// Mitsubishi GX Works2 project: 6.14 finsh   PLC: FX3G

// global labels: Global1
VAR_GLOBAL
  sw7_startday AT X007 : BOOL;
  output7_light AT Y007 : BOOL;
  sw5_emrgency AT X005 : BOOL;
  raw_matirial_end AT M1 : BOOL;
  matirial_end AT M1 : BOOL;
  output5_light AT M7 : BOOL;
  work_day_m5 AT M5 : BOOL;
  lamf_work_day AT Y007 : BOOL;
  Petel_input_amount AT D1148 : REAL;
  Petel_cornt_amount AT D1250 : REAL;
  Limonl_input_amount AT D1195 : REAL;
  Gomi_input_amount AT D1245 : REAL;
  Gomi_cornt_amount AT D1270 : REAL;
  Meatzv_input_amount AT D1295 : REAL;
  Meyatzev_input_amount AT D1295 : REAL;
  Meyatzev_cornt_amount AT D1300 : REAL;
  output AT D8282 : INT;
  start_ice_crem AT X001 : BOOL;
  timer_icecream5 AT TC1 : BOOL;
END_VAR
VAR_GLOBAL CONSTANT
  Sec_icecream : INT := K50;
END_VAR
VAR_GLOBAL
  start_icecream AT X001 : BOOL;
  Petel_ragil_help AT M52 : BOOL;
  Petel_pinoc_help AT M53 : BOOL;
  Limon_ragil_help AT M54 : BOOL;
  Limon_input_amount AT D1195 : REAL;
  Limon_cornt_amount AT D1200 : REAL;
  Limon_pinoc_help AT M55 : BOOL;
  Petel_ragil AT M22 : BOOL;
  Petel_pinoc AT M23 : BOOL;
  Limon_ragil AT M24 : BOOL;
  Limon_pinoc AT M25 : BOOL;
  lamp_y2 AT Y002 : BOOL;
END_VAR
VAR_GLOBAL CONSTANT
  division_constant : REAL := 400;
END_VAR
VAR_GLOBAL
  analog_input_1 AT D8280 : INT;
  goomigum_type AT D1502 : REAL;
  Min_regular AT E0.0 : REAL;
  Max_regular AT E5.0 : REAL;
  Min_pinuk AT E6.0 : REAL;
  check_inventory AT M20 : BOOL;
  choose_regular AT M300 : BOOL;
  choose_pinuk AT M400 : BOOL;
END_VAR
VAR_GLOBAL CONSTANT
  const280 : REAL := 280;
  const_280 : REAL := 280;
  conat_35 : REAL := 280;
  const_35 : REAL := 35;
END_VAR
VAR_GLOBAL
  not_petel_ragil AT M61 : BOOL;
END_VAR
VAR_GLOBAL CONSTANT
  const_385 : REAL := 385;
  const_105 : REAL := 105;
  const_70 : REAL := 70;
  const_0 : REAL;
  const_420 : REAL := 420;
END_VAR
VAR_GLOBAL
  not_Petel_pinoc AT M62 : BOOL;
  not_Limon_ragil AT M63 : BOOL;
END_VAR
VAR_GLOBAL CONSTANT
  const_560 : REAL := 560;
END_VAR
VAR_GLOBAL
  not_Limon_pinoc AT M64 : BOOL;
END_VAR
VAR_GLOBAL CONSTANT
  const_140 : REAL := 140;
END_VAR
VAR_GLOBAL
  check_matirial AT M4 : BOOL;
  work : BOOL;
END_VAR
VAR_GLOBAL CONSTANT
  Five_Sec_icecream : INT := 50;
END_VAR
VAR_GLOBAL
  Time_icecream_finish AT TS1 : BOOL;
  is_making_icecream AT Y000 : BOOL;
  start_freeze AT X002 : BOOL;
END_VAR
VAR_GLOBAL CONSTANT
  const_700 : REAL := 700;
  const_490 : REAL := 490;
  const_350 : REAL := 350;
END_VAR
VAR_GLOBAL
  Premium_petel_icecream AT D1190 : REAL;
  Premium_lemonl_icecream AT D1210 : REAL;
  Regular_petel_icecream AT D1230 : REAL;
  Regular_lemonl_icecream AT D1240 : REAL;
END_VAR
VAR_GLOBAL CONSTANT
  const_8 : REAL := 8;
  const_10 : REAL;
END_VAR
VAR_GLOBAL
  sen_10 AT X003 : BOOL;
  lemf_y2 AT Y002 : BOOL;
  lamf_y2 AT Y002 : BOOL;
  Start_Packing AT X004 : BOOL;
  first_packing AT X000 : BOOL;
END_VAR
VAR_GLOBAL CONSTANT
  couter_seven_cones : INT := 7;
END_VAR
VAR_GLOBAL
  done_seven AT CC1 : BOOL;
  finish_seven AT CS1 : BOOL;
END_VAR
VAR_GLOBAL CONSTANT
  const_1 : INT := 1;
END_VAR
VAR_GLOBAL
  current_counter_cones AT CN1 : INT;
END_VAR
VAR_GLOBAL CONSTANT
  const_6_word : INT := 6;
END_VAR
VAR_GLOBAL
  lamp_y4 AT Y004 : BOOL;
  Amount_packages AT D1160 : REAL;
END_VAR
VAR_GLOBAL CONSTANT
  ADD_Package : REAL := 1;
END_VAR
VAR_GLOBAL
  end_day AT M10 : BOOL;
END_VAR
VAR_GLOBAL CONSTANT
  MUL40 : REAL := 40;
END_VAR
VAR_GLOBAL
  OutputMul AT D1170 : REAL;
  Frozen_premium_petel AT D3030 : REAL;
  Frozen_premium_lemon AT D3020 : REAL;
  Frozen_regular_petel AT D3040 : REAL;
  Frozen_regular_lemon AT D3060 : REAL;
  Stir_premium_petel AT D3080 : REAL;
  Stir_premium_lemon AT D4000 : REAL;
  Gummy_to_prod AT D5000 : REAL;
  Stir_regular_petel AT D4020 : REAL;
  Stir_regular_lemon AT D4040 : REAL;
END_VAR
VAR_GLOBAL CONSTANT
  const_28 : REAL := 28;
END_VAR
VAR_GLOBAL
  start_blink AT M60 : BOOL;
  timer_reset AT M0 : BOOL;
END_VAR
VAR_GLOBAL CONSTANT
  const_5 : INT := 50;
END_VAR
VAR_GLOBAL
  End_Timer1 AT TS1 : BOOL;
  Blink1 AT Y005 : BOOL;
  End_Timer2 AT TS2 : BOOL;
  Timer2 AT TC2 : BOOL;
  Blink2 AT Y006 : BOOL;
END_VAR
VAR_GLOBAL CONSTANT
  const_3 : INT := 30;
END_VAR
VAR_GLOBAL
  raw_materialsl_ferm AT D1165 : REAL;
  timer8 AT TC3 : BOOL;
  END_Timer3 AT TS3 : BOOL;
  ragil AT M30 : BOOL;
  ragi AT M22 : BOOL;
  pinoc AT M40 : BOOL;
  pinuk AT M40 : BOOL;
  regular AT M30 : BOOL;
  Ts5 AT Y005 : BOOL;
  ts6 AT Y006 : BOOL;
  ts7 AT Y007 : BOOL;
  ts4 AT Y004 : BOOL;
  lemon_icecream AT D1240 : REAL;
  petel_icecream AT D1230 : REAL;
  Frozen_petel AT D3030 : REAL;
  Frozen_lemon AT D3040 : REAL;
  lemonl_icecream AT D1210 : REAL;
END_VAR
VAR_GLOBAL CONSTANT
  const_2000 : REAL := 2000;
  const_80 : INT := 80;
END_VAR
VAR_GLOBAL
  Stir_petel AT D4030 : REAL;
  Stir_lemon AT D4040 : REAL;
  check666 AT X006 : BOOL;
  Timer4 AT TC4 : BOOL;
  End_Timer4 AT TS4 : BOOL;
  Timer800 AT TC10 : BOOL;
  End_Timer800 AT TS10 : BOOL;
  Timer5007 AT TC20 : BOOL;
  End_Timer5007 AT TS20 : BOOL;
  Timer5 AT TC30 : BOOL;
  Timer500 AT TC50 : BOOL;
  End_Timer500 AT TS50 : BOOL;
  End_Timer5 AT TS30 : BOOL;
  time_reset AT TC1 : BOOL;
END_VAR
VAR_GLOBAL CONSTANT
  stamtimer : INT := 10;
END_VAR
VAR_GLOBAL
  stammmm AT TC8 : BOOL;
  StAm AT TS8 : BOOL;
END_VAR
VAR_GLOBAL CONSTANT
  MUL400 : REAL := 400;
END_VAR
VAR_GLOBAL
  timer_pinuk AT TC55 : BOOL;
  timer_regular AT TC33 : BOOL;
  AD_matay1 AT TS33 : BOOL;
  AD_matay2 AT TS55 : BOOL;
END_VAR
VAR_GLOBAL CONSTANT
  const_imashelhazona : INT := 30;
END_VAR
VAR_GLOBAL
  regular_blink AT TS33 : BOOL;
  pinuk_blink AT TS55 : BOOL;
END_VAR
VAR_GLOBAL CONSTANT
  const_05 : INT := 5;
END_VAR
VAR_GLOBAL
  count_reset AT M20 : BOOL;
  count_reset11 AT TC8 : BOOL;
END_VAR
VAR_GLOBAL CONSTANT
  const_10a : INT := 10;
END_VAR
VAR_GLOBAL
  reset11a AT TS8 : BOOL;
  delete_frozen AT M39 : BOOL;
  Time_to_blink AT TC15 : BOOL;
END_VAR
VAR_GLOBAL CONSTANT
  const_6 : INT := 60;
END_VAR
VAR_GLOBAL
  Time_to_blink_f AT TS15 : BOOL;
  lamf_blink_help AT M70 : BOOL;
  fictive_1 AT TC11 : BOOL;
  fictive_2 AT TC12 : BOOL;
  fictive_1_help AT TS11 : BOOL;
  fictive_2_help AT TS12 : BOOL;
  Finish_blink AT M11 : BOOL;
END_VAR

// task Task_01 (event TRUE, interval 0, priority 31): POU_01

PROGRAM POU_01
(* structured ladder/FBD written out as ST: instructions are called as NAME(EN, inputs, outputs); _pN, _eN, _tN stand for wires *)
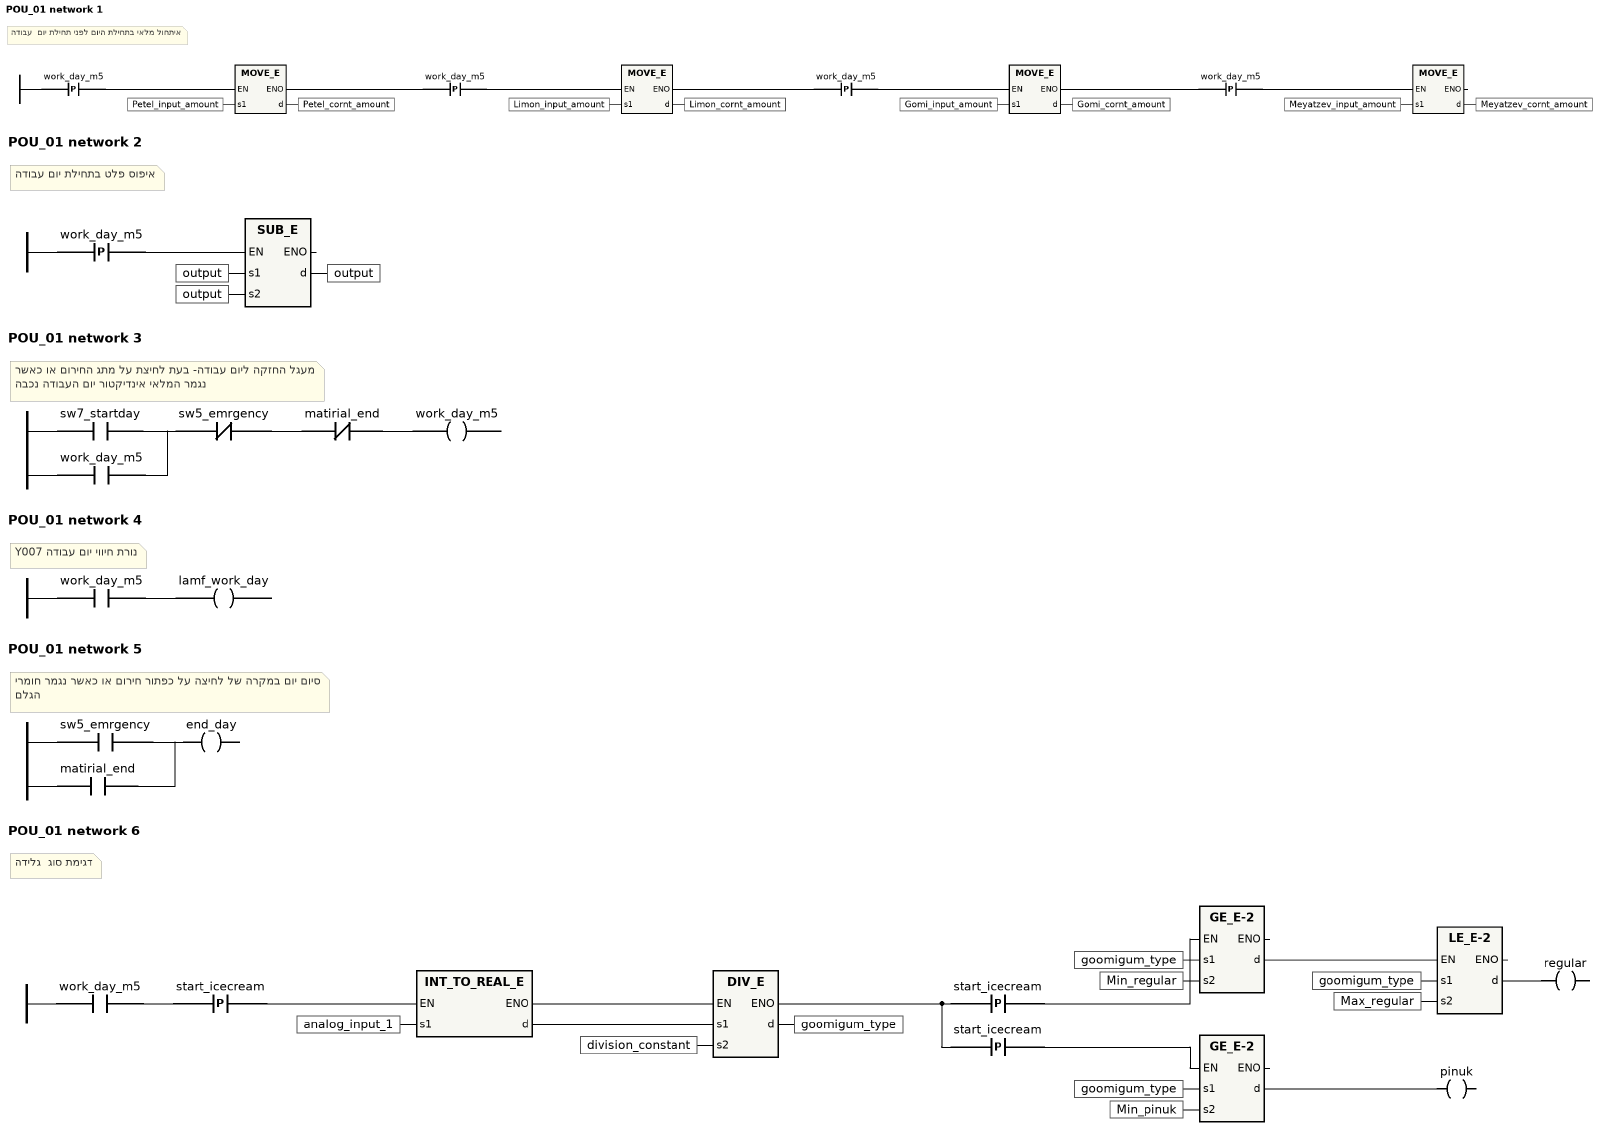
(* network 1 *)
(* איתחול מלאי בתחילת היום לפני תחילת יום  עבודה *)
_e1 := MOVE_E(LDP(TRUE, work_day_m5), Petel_input_amount, Petel_cornt_amount);
_e2 := MOVE_E(_e1 AND LDP(TRUE, work_day_m5), Limon_input_amount, Limon_cornt_amount);
_e3 := MOVE_E(_e2 AND LDP(TRUE, work_day_m5), Gomi_input_amount, Gomi_cornt_amount);
MOVE_E(_e3 AND LDP(TRUE, work_day_m5), Meyatzev_input_amount, Meyatzev_cornt_amount);
(* network 2 *)
(* איפוס פלט בתחילת יום עבודה *)
SUB_E(LDP(TRUE, work_day_m5), output, output, output);
(* network 3 *)
(* מעגל החזקה ליום עבודה- בעת לחיצת על מתג החירום או כאשר נגמר המלאי אינדיקטור יום העבודה נכבה *)
work_day_m5 := ((sw7_startday OR work_day_m5) AND NOT sw5_emrgency) AND NOT matirial_end;
(* network 4 *)
(* נורת חיווי יום עבודה Y007 *)
lamf_work_day := work_day_m5;
(* network 5 *)
(* סיום יום במקרה של לחיצה על כפתור חירום או כאשר נגמר חומרי הגלם *)
end_day := sw5_emrgency OR matirial_end;
(* network 6 *)
(* דגימת סוג  גלידה *)
_e2 := INT_TO_REAL_E(work_day_m5 AND LDP(TRUE, start_icecream), analog_input_1, _t1);
_e3 := DIV_E(_e2, _t1, division_constant, goomigum_type);
GE_E(_e3 AND LDP(TRUE, start_icecream), goomigum_type, Min_regular, _t4);
LE_E(_t4, goomigum_type, Max_regular, _t5);
regular := _t5;
GE_E(_e3 AND LDP(TRUE, start_icecream), goomigum_type, Min_pinuk, _t6);
pinuk := _t6;
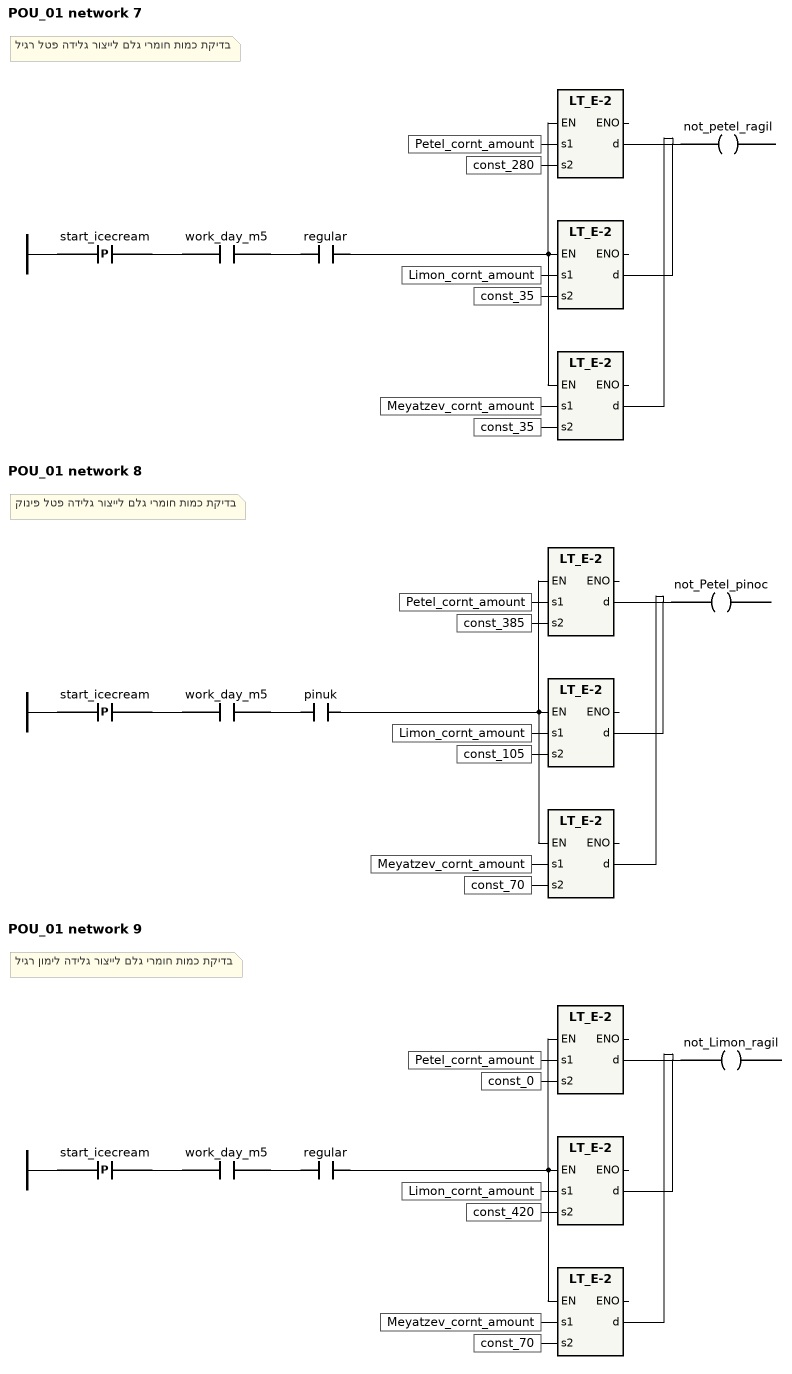
(* network 7 *)
(* בדיקת כמות חומרי גלם לייצור גלידה פטל רגיל *)
_p1 := LDP(TRUE, start_icecream) AND work_day_m5 AND regular;
LT_E(_p1, Petel_cornt_amount, const_280, _t2);
LT_E(_p1, Limon_cornt_amount, const_35, _t3);
LT_E(_p1, Meyatzev_cornt_amount, const_35, _t4);
not_petel_ragil := _t2 OR _t3 OR _t4;
(* network 8 *)
(* בדיקת כמות חומרי גלם לייצור גלידה פטל פינוק *)
_p1 := LDP(TRUE, start_icecream) AND work_day_m5 AND pinuk;
LT_E(_p1, Petel_cornt_amount, const_385, _t2);
LT_E(_p1, Limon_cornt_amount, const_105, _t3);
LT_E(_p1, Meyatzev_cornt_amount, const_70, _t4);
not_Petel_pinoc := _t2 OR _t3 OR _t4;
(* network 9 *)
(* בדיקת כמות חומרי גלם לייצור גלידה לימון רגיל *)
_p1 := LDP(TRUE, start_icecream) AND work_day_m5 AND regular;
LT_E(_p1, Petel_cornt_amount, const_0, _t2);
LT_E(_p1, Limon_cornt_amount, const_420, _t3);
LT_E(_p1, Meyatzev_cornt_amount, const_70, _t4);
not_Limon_ragil := _t2 OR _t3 OR _t4;
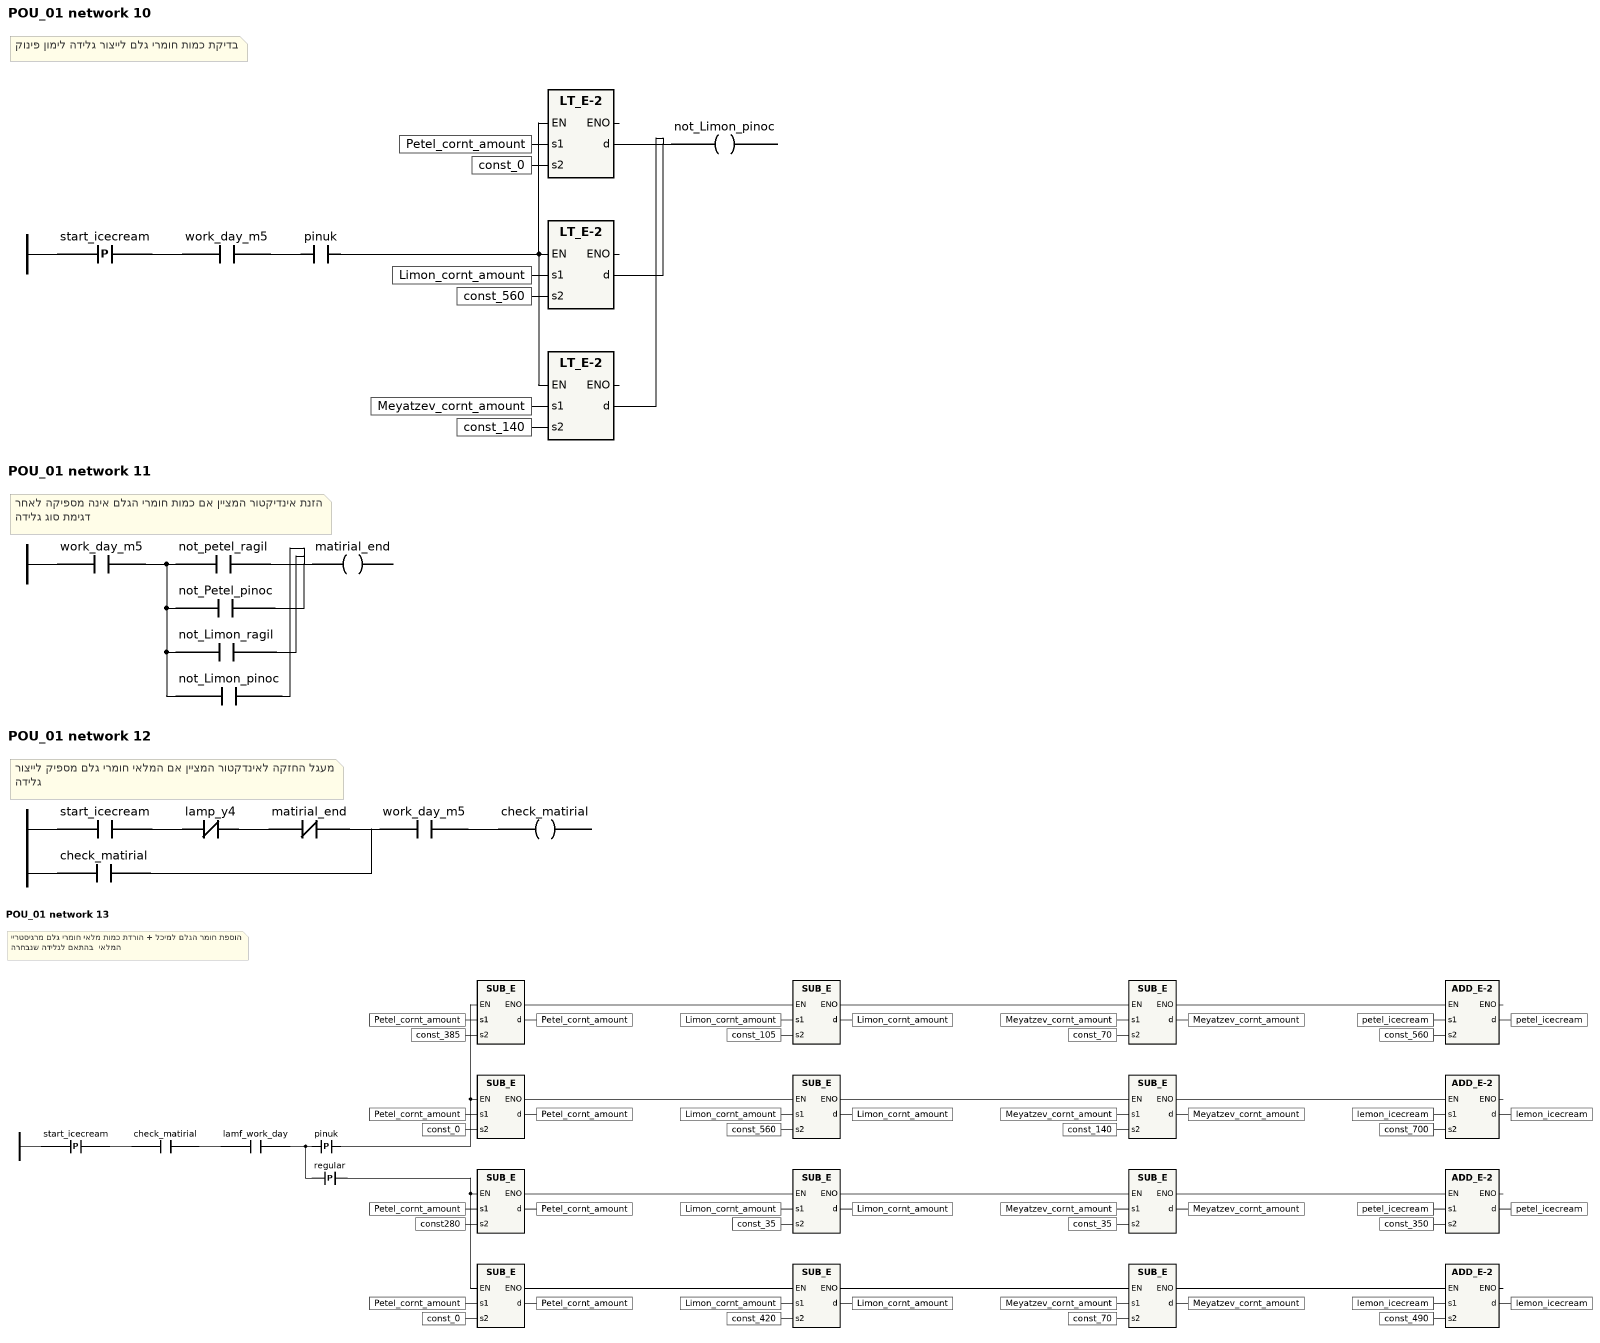
(* network 10 *)
(* בדיקת כמות חומרי גלם לייצור גלידה לימון פינוק *)
_p1 := LDP(TRUE, start_icecream) AND work_day_m5 AND pinuk;
LT_E(_p1, Petel_cornt_amount, const_0, _t2);
LT_E(_p1, Limon_cornt_amount, const_560, _t3);
LT_E(_p1, Meyatzev_cornt_amount, const_140, _t4);
not_Limon_pinoc := _t2 OR _t3 OR _t4;
(* network 11 *)
(* הזנת אינדיקטור המציין אם כמות חומרי הגלם אינה מספיקה לאחר דגימת סוג גלידה *)
matirial_end := (work_day_m5 AND not_petel_ragil) OR (work_day_m5 AND not_Petel_pinoc) OR (work_day_m5 AND not_Limon_ragil) OR (work_day_m5 AND not_Limon_pinoc);
(* network 12 *)
(* מעגל החזקה לאינדקטור המציין אם המלאי חומרי גלם מספיק לייצור גלידה *)
check_matirial := ((start_icecream AND NOT lamp_y4 AND NOT matirial_end) OR check_matirial) AND work_day_m5;
(* network 13 *)
(* הוספת חומר הגלם למיכל + הורדת כמות מלאי חומרי גלם מרגיסטריי המלאי  בהתאם לגלידה שנבחרה *)
_p1 := LDP(TRUE, start_icecream) AND check_matirial AND lamf_work_day;
_p2 := _p1 AND LDP(TRUE, pinuk);
_e3 := SUB_E(_p2, Petel_cornt_amount, const_385, Petel_cornt_amount);
_e4 := SUB_E(_e3, Limon_cornt_amount, const_105, Limon_cornt_amount);
_e5 := SUB_E(_e4, Meyatzev_cornt_amount, const_70, Meyatzev_cornt_amount);
ADD_E(_e5, petel_icecream, const_560, petel_icecream);
_e6 := SUB_E(_p2, Petel_cornt_amount, const_0, Petel_cornt_amount);
_e7 := SUB_E(_e6, Limon_cornt_amount, const_560, Limon_cornt_amount);
_e8 := SUB_E(_e7, Meyatzev_cornt_amount, const_140, Meyatzev_cornt_amount);
ADD_E(_e8, lemon_icecream, const_700, lemon_icecream);
_p9 := _p1 AND LDP(TRUE, regular);
_e10 := SUB_E(_p9, Petel_cornt_amount, const280, Petel_cornt_amount);
_e11 := SUB_E(_e10, Limon_cornt_amount, const_35, Limon_cornt_amount);
_e12 := SUB_E(_e11, Meyatzev_cornt_amount, const_35, Meyatzev_cornt_amount);
ADD_E(_e12, petel_icecream, const_350, petel_icecream);
_e13 := SUB_E(_p9, Petel_cornt_amount, const_0, Petel_cornt_amount);
_e14 := SUB_E(_e13, Limon_cornt_amount, const_420, Limon_cornt_amount);
_e15 := SUB_E(_e14, Meyatzev_cornt_amount, const_70, Meyatzev_cornt_amount);
ADD_E(_e15, lemon_icecream, const_490, lemon_icecream);
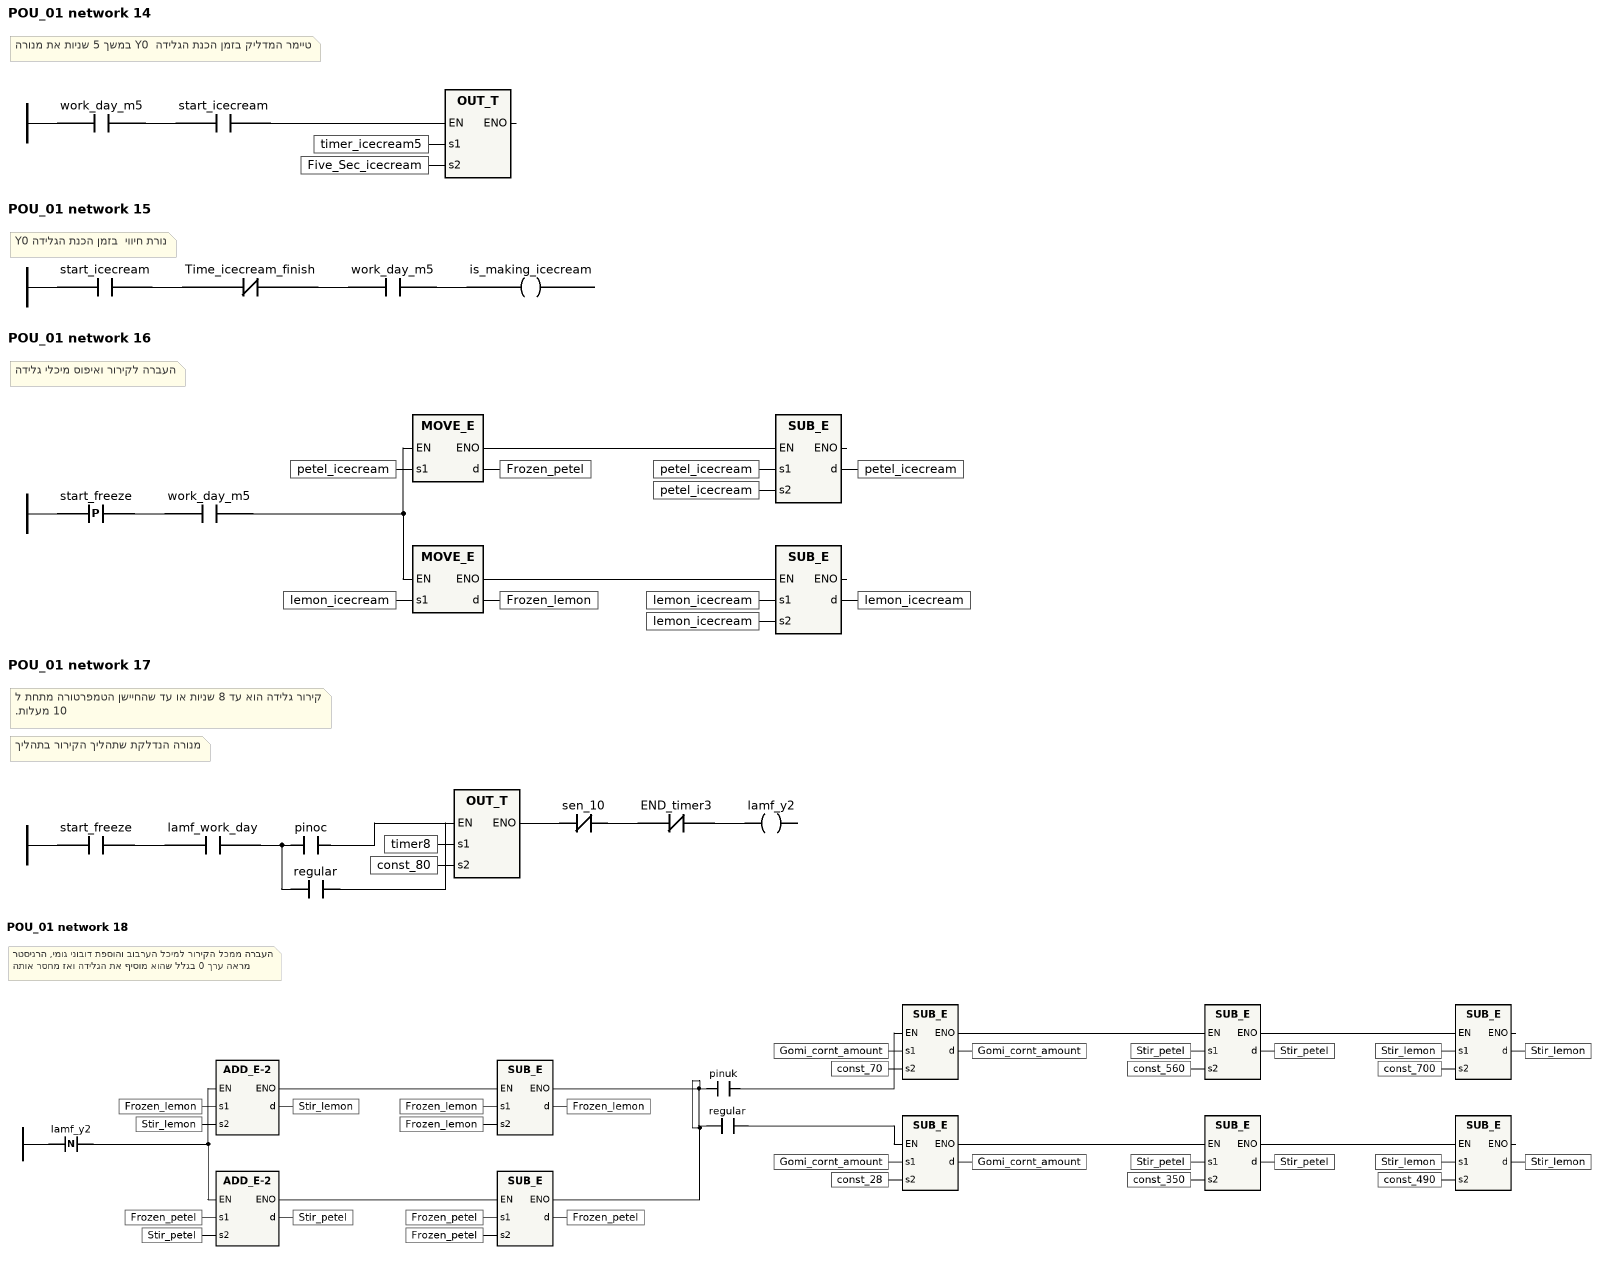
(* network 14 *)
(* טיימר המדליק בזמן הכנת הגלידה  Y0 במשך 5 שניות את מנורה *)
OUT_T(work_day_m5 AND start_icecream, timer_icecream5, Five_Sec_icecream);
(* network 15 *)
(* נורת חיווי  בזמן הכנת הגלידה Y0 *)
is_making_icecream := start_icecream AND NOT Time_icecream_finish AND work_day_m5;
(* network 16 *)
(* העברה לקירור ואיפוס מיכלי גלידה *)
_p1 := LDP(TRUE, start_freeze) AND work_day_m5;
_e2 := MOVE_E(_p1, petel_icecream, Frozen_petel);
SUB_E(_e2, petel_icecream, petel_icecream, petel_icecream);
_e3 := MOVE_E(_p1, lemon_icecream, Frozen_lemon);
SUB_E(_e3, lemon_icecream, lemon_icecream, lemon_icecream);
(* network 17 *)
(* קירור גלידה הוא עד 8 שניות או עד שהחיישן הטמפרטורה מתחת ל 10 מעלות. *)
(* מנורה הנדלקת שתהליך הקירור בתהליך *)
_p1 := start_freeze AND lamf_work_day;
_e2 := OUT_T((_p1 AND pinoc) OR (_p1 AND regular), timer8, const_80);
lamf_y2 := _e2 AND NOT sen_10 AND NOT END_timer3;
(* network 18 *)
(* העברה ממכל הקירור למיכל הערבוב והוספת דובוני גומי, הרגיסטר מראה ערך 0 בגלל שהוא מוסיף את הגלידה ואז מחסר אותה *)
_p1 := LDF(TRUE, lamf_y2);
_e2 := ADD_E(_p1, Frozen_lemon, Stir_lemon, Stir_lemon);
_e3 := SUB_E(_e2, Frozen_lemon, Frozen_lemon, Frozen_lemon);
_e4 := ADD_E(_p1, Frozen_petel, Stir_petel, Stir_petel);
_e5 := SUB_E(_e4, Frozen_petel, Frozen_petel, Frozen_petel);
_p6 := _e3 OR _e5;
_e7 := SUB_E(_p6 AND pinuk, Gomi_cornt_amount, const_70, Gomi_cornt_amount);
_e8 := SUB_E(_e7, Stir_petel, const_560, Stir_petel);
SUB_E(_e8, Stir_lemon, const_700, Stir_lemon);
_e9 := SUB_E(_p6 AND regular, Gomi_cornt_amount, const_28, Gomi_cornt_amount);
_e10 := SUB_E(_e9, Stir_petel, const_350, Stir_petel);
SUB_E(_e10, Stir_lemon, const_490, Stir_lemon);
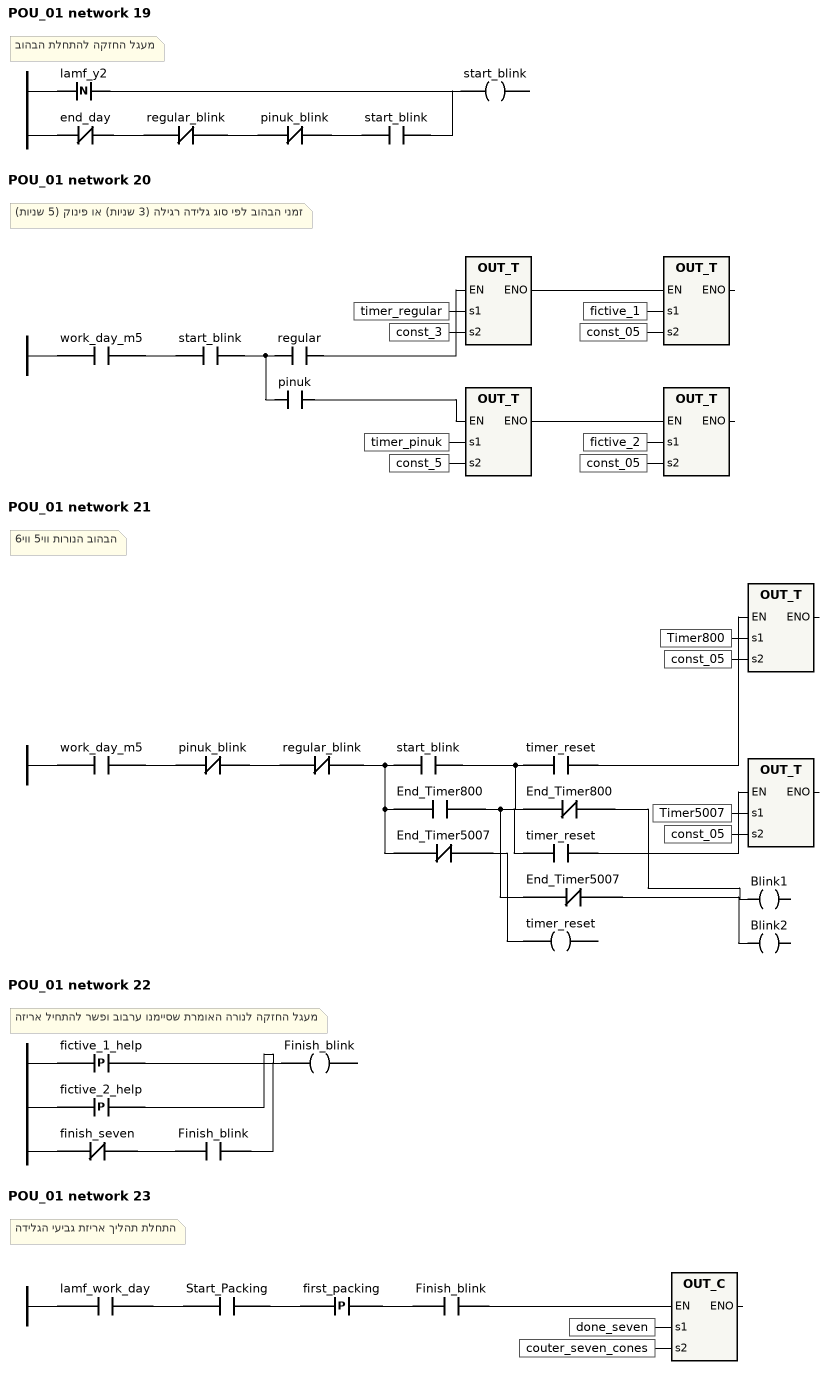
(* network 19 *)
(* מעגל החזקה להתחלת הבהוב *)
start_blink := LDF(TRUE, lamf_y2) OR (NOT end_day AND NOT regular_blink AND NOT pinuk_blink AND start_blink);
(* network 20 *)
(* זמני הבהוב לפי סוג גלידה רגילה (3 שניות) או פינוק (5 שניות) *)
_p1 := work_day_m5 AND start_blink;
_e2 := OUT_T(_p1 AND regular, timer_regular, const_3);
OUT_T(_e2, fictive_1, const_05);
_e3 := OUT_T(_p1 AND pinuk, timer_pinuk, const_5);
OUT_T(_e3, fictive_2, const_05);
(* network 21 *)
(* הבהוב הנורות ווי5 ווי6 *)
_p1 := work_day_m5 AND NOT pinuk_blink AND NOT regular_blink;
_p2 := _p1 AND start_blink;
OUT_T(_p2 AND timer_reset, Timer800, const_05);
Blink1 := _p2 AND NOT End_Timer800;
_p3 := _p1 AND End_Timer800;
OUT_T(_p3 AND timer_reset, Timer5007, const_05);
Blink2 := _p3 AND NOT End_Timer5007;
timer_reset := _p1 AND NOT End_Timer5007;
(* network 22 *)
(* מעגל החזקה לנורה האומרת שסיימנו ערבוב ופשר להתחיל אריזה *)
Finish_blink := LDP(TRUE, fictive_1_help) OR LDP(TRUE, fictive_2_help) OR (NOT finish_seven AND Finish_blink);
(* network 23 *)
(* התחלת תהליך אריזת גביעי הגלידה *)
OUT_C(lamf_work_day AND Start_Packing AND LDP(TRUE, first_packing) AND Finish_blink, done_seven, couter_seven_cones);
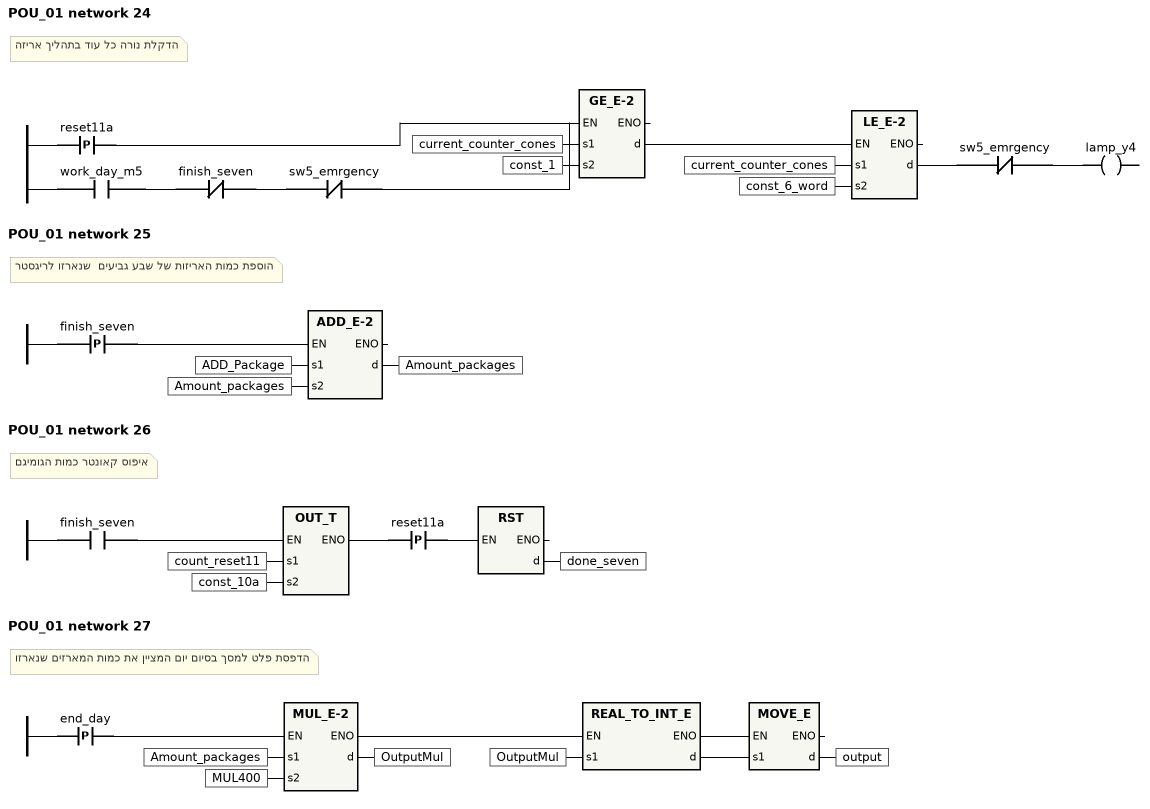
(* network 24 *)
(* הדקלת נורה כל עוד בתהליך אריזה *)
GE_E(LDP(TRUE, reset11a) OR (work_day_m5 AND NOT finish_seven AND NOT sw5_emrgency), current_counter_cones, const_1, _t1);
LE_E(_t1, current_counter_cones, const_6_word, _t2);
lamp_y4 := _t2 AND NOT sw5_emrgency;
(* network 25 *)
(* הוספת כמות האריזות של שבע גביעים  שנארזו לריגסטר *)
ADD_E(LDP(TRUE, finish_seven), ADD_Package, Amount_packages, Amount_packages);
(* network 26 *)
(* איפוס קאונטר כמות הגומיגם *)
_e1 := OUT_T(finish_seven, count_reset11, const_10a);
RST(_e1 AND LDP(TRUE, reset11a), done_seven);
(* network 27 *)
(* הדפסת פלט למסך בסיום יום המציין את כמות המארזים שנארזו *)
_e1 := MUL_E(LDP(TRUE, end_day), Amount_packages, MUL400, OutputMul);
_e3 := REAL_TO_INT_E(_e1, OutputMul, _t2);
MOVE_E(_e3, _t2, output);
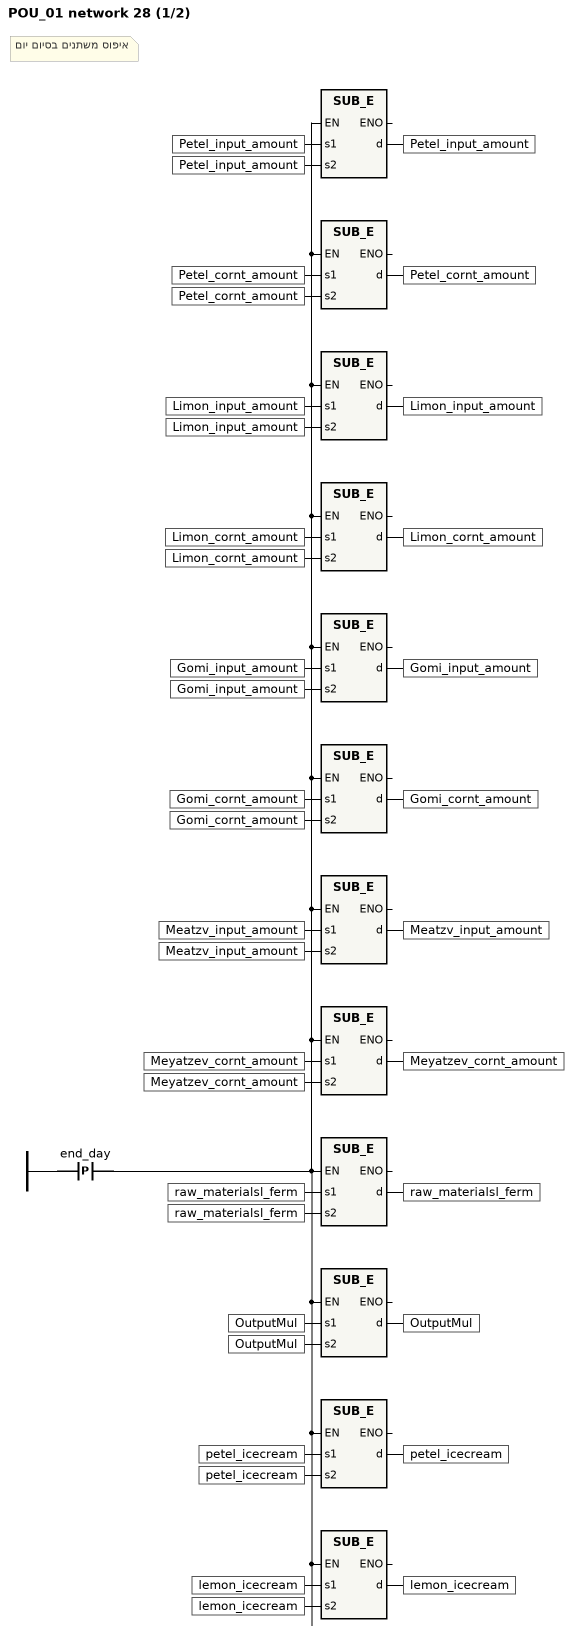
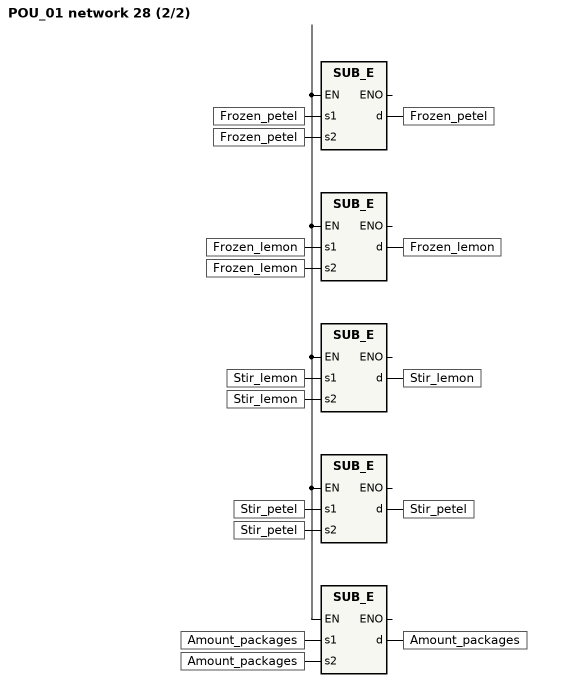
(* network 28 *)
(* איפוס משתנים בסיום יום *)
_p1 := LDP(TRUE, end_day);
SUB_E(_p1, Petel_input_amount, Petel_input_amount, Petel_input_amount);
SUB_E(_p1, Petel_cornt_amount, Petel_cornt_amount, Petel_cornt_amount);
SUB_E(_p1, Limon_input_amount, Limon_input_amount, Limon_input_amount);
SUB_E(_p1, Limon_cornt_amount, Limon_cornt_amount, Limon_cornt_amount);
SUB_E(_p1, Gomi_input_amount, Gomi_input_amount, Gomi_input_amount);
SUB_E(_p1, Gomi_cornt_amount, Gomi_cornt_amount, Gomi_cornt_amount);
SUB_E(_p1, Meatzv_input_amount, Meatzv_input_amount, Meatzv_input_amount);
SUB_E(_p1, Meyatzev_cornt_amount, Meyatzev_cornt_amount, Meyatzev_cornt_amount);
SUB_E(_p1, raw_materialsl_ferm, raw_materialsl_ferm, raw_materialsl_ferm);
SUB_E(_p1, OutputMul, OutputMul, OutputMul);
SUB_E(_p1, petel_icecream, petel_icecream, petel_icecream);
SUB_E(_p1, lemon_icecream, lemon_icecream, lemon_icecream);
SUB_E(_p1, Frozen_petel, Frozen_petel, Frozen_petel);
SUB_E(_p1, Frozen_lemon, Frozen_lemon, Frozen_lemon);
SUB_E(_p1, Stir_lemon, Stir_lemon, Stir_lemon);
SUB_E(_p1, Stir_petel, Stir_petel, Stir_petel);
SUB_E(_p1, Amount_packages, Amount_packages, Amount_packages);
END_PROGRAM
